// TIA Portal V18 export
VAR_GLOBAL   // PLC tag table "AO"
   "H/SSR_019_CV01_CVOUT" AT %QW26 : Int;
   "H/SSR_019_CV02_CVOUT" AT %QW28 : Int;
   "H/SSR_019_CV03_CVOUT" AT %QW30 : Int;
   SPARE AT %QW38 : Int;
   SPARE_1 AT %QW40 : Int;
   SPARE_2 AT %QW42 : Int;
   SPARE_3 AT %QW44 : Int;
   SPARE_4 AT %QW46 : Int;
   SPARE_5 AT %QW48 : Int;
   SPARE_6 AT %QW50 : Int;
   SPARE_7 AT %QW52 : Int;
   SPARE_8 AT %QW54 : Int;
   SPARE_9 AT %QW56 : Int;
   SPARE_10 AT %QW58 : Int;
   SPARE_11 AT %QW60 : Int;
   SPARE_12 AT %QW62 : Int;
   SPARE_13 AT %QW64 : Int;
   SPARE_14 AT %QW66 : Int;
END_VAR
